// TIA Portal V18 export
TYPE "RCS_SysAuto_V1"
   STRUCT
      Mode : Bool;   // Sation in Auto Mode (bit tag)
      Running : Bool;   // Sation in Auto Running Status
      RunningPause : Bool;   // Sation in Auto Running Pause (1=Runing, 0=Pause)
      RunningOver : Bool;   // Runing over (clear line or Station)
      StepMode : Bool;   // Sation in Step Mode
      OneCycleMode : Bool;   // Sation in One Cycle Mode
      StartAuto : Bool;   // Flow Start
      AllRun : Bool;   // All pm are running
      Status : Int;   // 0NotReady, 1Ready, 2AutoRunning, 3EStop, 4Alarm
   END_STRUCT;
END_TYPE
